// TIA Portal V18 export
DATA_BLOCK "ST10_CountCycleTimeMain_DB"   // DB1009
VERSION : 0.1
// stored: AutoNumber false, DBAccessibleFromOPCUA true, DBAccessibleFromWebserver true, InstanceOfName ST10_CountCycleTimeMain, InstanceOfType FB
"ST10_CountCycleTimeMain"
   // VAR_INPUT
   //    iAlwaysOn : Bool;
   //    iRun : Bool;
   //    iManualMode : Bool;
   //    iAutoMode : Bool;
   //    iAutoRunning : Bool;
   // END_VAR
   // VAR
   //    MianCountCycleTime { S7_SetPoint := 'True'} : "Count_CycleTime";
   //    PM1CountCycleTime { S7_SetPoint := 'True'} : "Count_CycleTime_V3";
   //    PM2CountCycleTime { S7_SetPoint := 'True'} : "Count_CycleTime_V3";
   //    PM3CountCycleTime { S7_SetPoint := 'True'} : "Count_CycleTime_V3";
   //    PM4CountCycleTime { S7_SetPoint := 'True'} : "Count_CycleTime_V3";
   //    PM5CountCycleTime { S7_SetPoint := 'True'} : "Count_CycleTime_V3";
   //    PM6CountCycleTime { S7_SetPoint := 'True'} : "Count_CycleTime_V3";
   //    PM7CountCycleTime { S7_SetPoint := 'True'} : "Count_CycleTime_V3";
   //    PM8CountCycleTime { S7_SetPoint := 'True'} : "Count_CycleTime_V3";
   //    PM9CountCycleTime { S7_SetPoint := 'True'} : "Count_CycleTime_V3";
   //    PM10CountCycleTime { S7_SetPoint := 'True'} : "Count_CycleTime_V3";
   //    PM11CountCycleTime { S7_SetPoint := 'True'} : "Count_CycleTime_V3";
   //    PM12CountCycleTime { S7_SetPoint := 'True'} : "Count_CycleTime_V3";
   //    PM13CountCycleTime { S7_SetPoint := 'True'} : "Count_CycleTime_V3";
   //    PM14CountCycleTime { S7_SetPoint := 'True'} : "Count_CycleTime_V3";
   //    PM15CountCycleTime { S7_SetPoint := 'True'} : "Count_CycleTime_V3";
   //    PM16CountCycleTime { S7_SetPoint := 'True'} : "Count_CycleTime_V3";
   //    PM17CountCycleTime { S7_SetPoint := 'True'} : "Count_CycleTime_V3";
   //    PM18CountCycleTime { S7_SetPoint := 'True'} : "Count_CycleTime_V3";
   //    PM19CountCycleTime { S7_SetPoint := 'True'} : "Count_CycleTime_V3";
   //    PM20CountCycleTime { S7_SetPoint := 'True'} : "Count_CycleTime_V3";
   //    PM21CountCycleTime { S7_SetPoint := 'True'} : "Count_CycleTime_V3";
   //    PM22CountCycleTime { S7_SetPoint := 'True'} : "Count_CycleTime_V3";
   //    PM23CountCycleTime { S7_SetPoint := 'True'} : "Count_CycleTime_V3";
   //    PM24CountCycleTime { S7_SetPoint := 'True'} : "Count_CycleTime_V3";
   //    PM25CountCycleTime { S7_SetPoint := 'True'} : "Count_CycleTime_V3";
   //    PM26CountCycleTime { S7_SetPoint := 'True'} : "Count_CycleTime_V3";
   //    PM27CountCycleTime { S7_SetPoint := 'True'} : "Count_CycleTime_V3";
   //    PM28CountCycleTime { S7_SetPoint := 'True'} : "Count_CycleTime_V3";
   //    PM29CountCycleTime { S7_SetPoint := 'True'} : "Count_CycleTime_V3";
   //    PM30CountCycleTime { S7_SetPoint := 'True'} : "Count_CycleTime_V3";
   // END_VAR
BEGIN
END_DATA_BLOCK
